(* Schneider Machine Expert - Basic project Tank_Level_RTD_v29, file version 3.0.0.0 *)
(* ProjectInformations: Name=New project *)

HARDWARE
  Cpu 0: TM221CE40T
  ModuleExtensionObject 0: TM3TI4/G
  EthernetConfiguration: NetworkName=M221, IpAllocationMode=FixedAddress, IpAddress=0.0.0.0, SubnetMask=0.0.0.0
  EthernetConfiguration: NetworkName=M221, IpAllocationMode=FixedAddress, IpAddress=0.0.0.0, SubnetMask=0.0.0.0
  EthernetConfiguration: NetworkName=M221, IpAllocationMode=FixedAddress, IpAddress=0.0.0.0, SubnetMask=0.0.0.0
  SerialLineConfiguration: Baud=Baud19200, Parity=ParityEven, DataBits=DataBits8, StopBits=StopBits1, PhysicalMedium=PhysicalMediumRs485, TransmissionMode=TransmissionModeModbusRtu, SlaveId=1, Addressing=SlaveAddressing
  MastTask: UsePeriodScanMode=false, PeriodScan=100
  FastTask: Period=255
  CpuBehavior: StartingMode=StartAsPreviousState, AutoSaveRamOnEeprom=true, WatchdogPeriod=250

SYMBOLS  (address, symbol, comment, settings)
  %M0       SYSTEM_READY
  %M1       TANK_LEVEL_LOW
  %M2       TANK_LEVEL_HIGH
  %S0       SB_COLDSTART  "Indicates or executes a cold start (data initialized to default values)"
  %S1       SB_WARMSTART  "Indicates there was a warm start with data backup"
  %TM0        [Preset=3, Base=OneSecond]
  %I0.0     EMERGENCY_PB
  %IW0.0      [Type=Type_0_10V, Scope=Scope_Normal, Minimum=0, Maximum=1000]
  %IW1.0    RTD_TEMP  [Type=Type_NotUsed, Scope=Scope_NotUsed, Minimum=0, Maximum=0]

POU New POU
  (* SectionNumber=0 *)

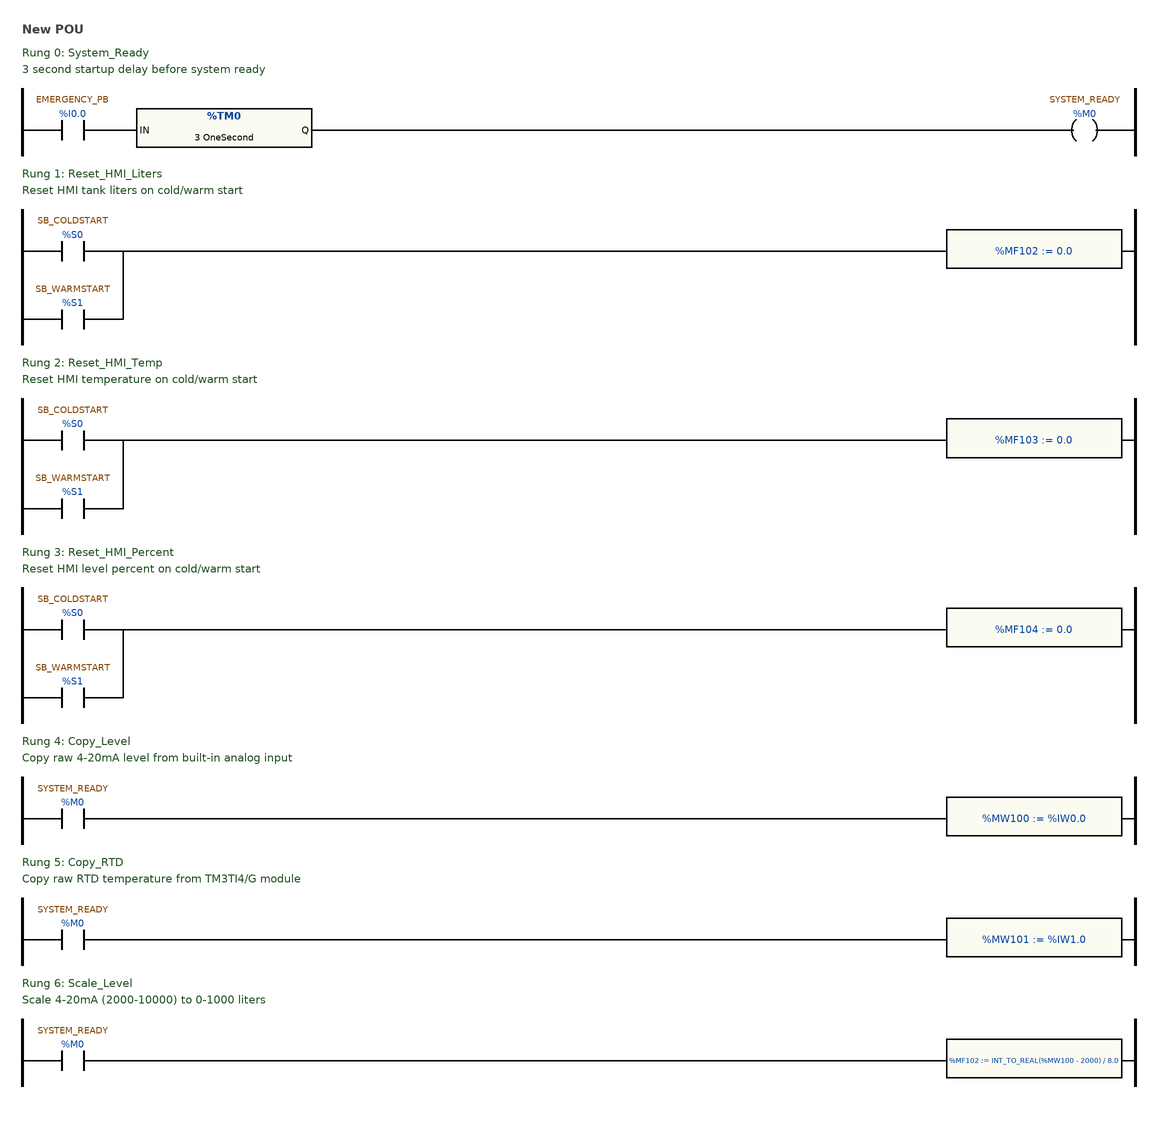

// Rung 0: System_Ready
// 3 second startup delay before system ready
  BLK %TM0
  LD %I0.0                (* EMERGENCY_PB *)
  IN
  OUT_BLK
  LD Q
  ST %M0                  (* SYSTEM_READY *)
  END_BLK
  // as ST:
  //   %TM0(IN := EMERGENCY_PB);
  //   SYSTEM_READY := %TM0.Q;

// Rung 1: Reset_HMI_Liters
// Reset HMI tank liters on cold/warm start
  LD %S0                  (* SB_COLDSTART *)
  OR %S1                  (* SB_WARMSTART *)
  [ %MF102 := 0.0 ]
  // %S0: Cold start
  // %S1: Warm start
  // as ST:
  //   IF SB_COLDSTART OR SB_WARMSTART THEN %MF102 := 0.0; END_IF;

// Rung 2: Reset_HMI_Temp
// Reset HMI temperature on cold/warm start
  LD %S0                  (* SB_COLDSTART *)
  OR %S1                  (* SB_WARMSTART *)
  [ %MF103 := 0.0 ]
  // %S0: Cold start
  // %S1: Warm start
  // as ST:
  //   IF SB_COLDSTART OR SB_WARMSTART THEN %MF103 := 0.0; END_IF;

// Rung 3: Reset_HMI_Percent
// Reset HMI level percent on cold/warm start
  LD %S0                  (* SB_COLDSTART *)
  OR %S1                  (* SB_WARMSTART *)
  [ %MF104 := 0.0 ]
  // %S0: Cold start
  // %S1: Warm start
  // as ST:
  //   IF SB_COLDSTART OR SB_WARMSTART THEN %MF104 := 0.0; END_IF;

// Rung 4: Copy_Level
// Copy raw 4-20mA level from built-in analog input
  LD %M0                  (* SYSTEM_READY *)
  [ %MW100 := %IW0.0 ]
  // as ST:
  //   IF SYSTEM_READY THEN %MW100 := %IW0.0; END_IF;

// Rung 5: Copy_RTD
// Copy raw RTD temperature from TM3TI4/G module
  LD %M0                  (* SYSTEM_READY *)
  [ %MW101 := %IW1.0 ]    (* RTD_TEMP *)
  // as ST:
  //   IF SYSTEM_READY THEN %MW101 := RTD_TEMP; END_IF;

// Rung 6: Scale_Level
// Scale 4-20mA (2000-10000) to 0-1000 liters
  LD %M0                  (* SYSTEM_READY *)
  [ %MF102 := INT_TO_REAL(%MW100 - 2000) / 8.0 ]
  // as ST:
  //   IF SYSTEM_READY THEN %MF102 := INT_TO_REAL(%MW100 - 2000) / 8.0; END_IF;

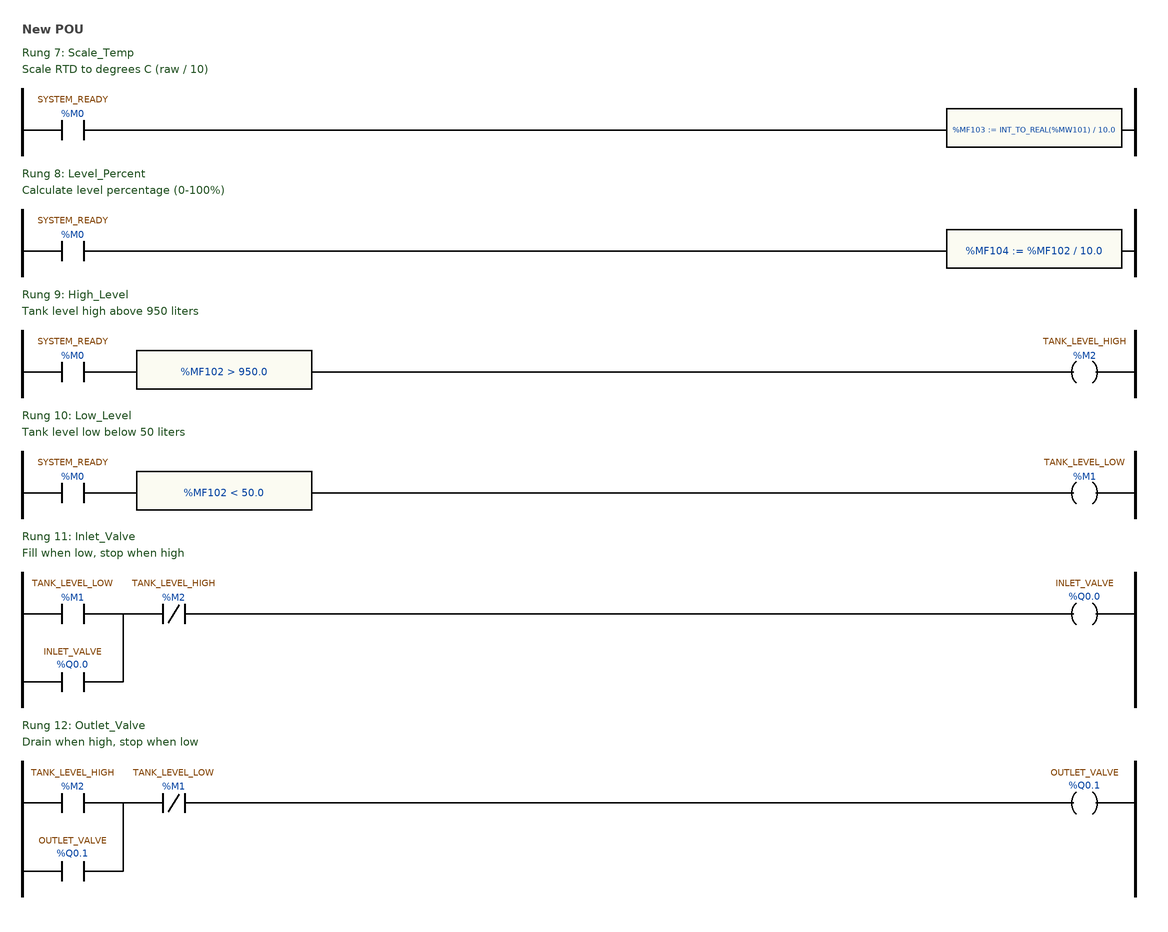

// Rung 7: Scale_Temp
// Scale RTD to degrees C (raw / 10)
  LD %M0                  (* SYSTEM_READY *)
  [ %MF103 := INT_TO_REAL(%MW101) / 10.0 ]
  // as ST:
  //   IF SYSTEM_READY THEN %MF103 := INT_TO_REAL(%MW101) / 10.0; END_IF;

// Rung 8: Level_Percent
// Calculate level percentage (0-100%)
  LD %M0                  (* SYSTEM_READY *)
  [ %MF104 := %MF102 / 10.0 ]
  // as ST:
  //   IF SYSTEM_READY THEN %MF104 := %MF102 / 10.0; END_IF;

// Rung 9: High_Level
// Tank level high above 950 liters
  LD %M0                  (* SYSTEM_READY *)
  AND [ %MF102 > 950.0 ]
  ST %M2                  (* TANK_LEVEL_HIGH *)
  // as ST:
  //   TANK_LEVEL_HIGH := SYSTEM_READY AND %MF102 > 950.0;

// Rung 10: Low_Level
// Tank level low below 50 liters
  LD %M0                  (* SYSTEM_READY *)
  AND [ %MF102 < 50.0 ]
  ST %M1                  (* TANK_LEVEL_LOW *)
  // as ST:
  //   TANK_LEVEL_LOW := SYSTEM_READY AND %MF102 < 50.0;

// Rung 11: Inlet_Valve
// Fill when low, stop when high
  LD %M1                  (* TANK_LEVEL_LOW *)
  OR %Q0.0
  ANDN %M2                (* TANK_LEVEL_HIGH *)
  ST %Q0.0
  // as ST:
  //   %Q0.0 := (TANK_LEVEL_LOW OR %Q0.0) AND NOT TANK_LEVEL_HIGH;

// Rung 12: Outlet_Valve
// Drain when high, stop when low
  LD %M2                  (* TANK_LEVEL_HIGH *)
  OR %Q0.1
  ANDN %M1                (* TANK_LEVEL_LOW *)
  ST %Q0.1
  // as ST:
  //   %Q0.1 := (TANK_LEVEL_HIGH OR %Q0.1) AND NOT TANK_LEVEL_LOW;
